(* IEC 61131-3 sources: volt/packages/volt-lsp-iec/test-corpus/bakon-nano/Device/Plc Logic/Application/Library Manager/SysTypes, 3 files *)

(* ---- RTS_IEC_HANDLE.dut ---- *)
TYPE RTS_IEC_HANDLE : POINTER TO BYTE;
END_TYPE

(* ---- RTS_IEC_RESULT.dut ---- *)
TYPE RTS_IEC_RESULT : UDINT;
END_TYPE

(* ---- HANDLECONSTANTS.gvl ---- *)
VAR_GLOBAL
	RTS_INVALID_HANDLE : RTS_IEC_HANDLE := 16#FFFFFFFF;
END_VAR
